// LS Electric XG5000 project: xg
// PLC NewPLC
// module base 0 slot 0: 입출력 모듈:XBC-DR32H (DC 24V 입력, 릴레이 출력 32점)
// module base 0 slot 1: 위치결정 모듈:XBF-PD02A (위치결정 펄스(LD)출력형, 2축)
// module base 0 slot 2: 출력 모듈:XBE-TN/TP16A (트랜지스터 출력, 16점 (싱크출력/소스출력))

PROGRAM NewProgram (task: 스캔 프로그램)

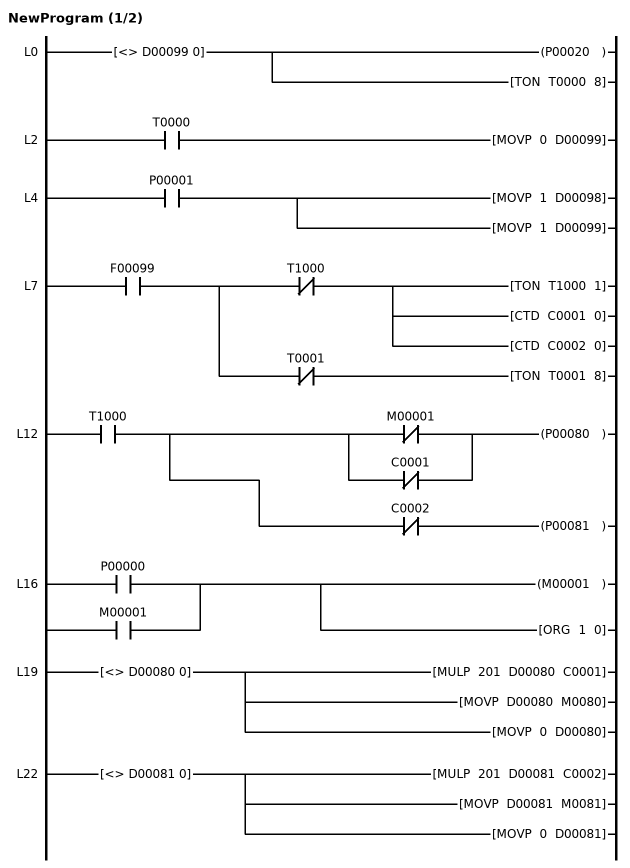
; L0
LOAD<>    D00099 0
OUT       P00020
TON       T0000 8
; L2
LOAD      T0000
MOVP      0 D00099
; L4
LOAD      P00001
MOVP      1 D00098
MOVP      1 D00099
; L7
LOAD      F00099
MPUSH
AND NOT   T1000
TON       T1000 1
CTD       C0001 0
CTD       C0002 0
MPOP
AND NOT   T0001
TON       T0001 8
; L12
LOAD      T1000
MPUSH
LOAD NOT  M00001
OR NOT    C0001
AND LOAD
OUT       P00080
MPOP
AND NOT   C0002
OUT       P00081
; L16
LOAD      P00000
OR        M00001
OUT       M00001
ORG       1 0
; L19
LOAD<>    D00080 0
MULP      201 D00080 C0001
MOVP      D00080 M0080
MOVP      0 D00080
; L22
LOAD<>    D00081 0
MULP      201 D00081 C0002
MOVP      D00081 M0081
MOVP      0 D00081

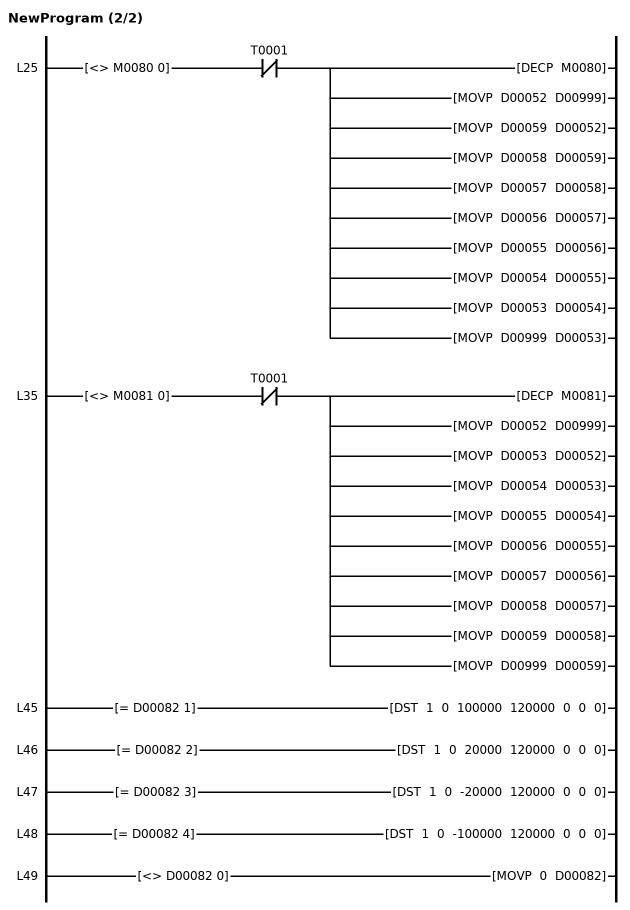
; L25
LOAD<>    M0080 0
AND NOT   T0001
DECP      M0080
MOVP      D00052 D00999
MOVP      D00059 D00052
MOVP      D00058 D00059
MOVP      D00057 D00058
MOVP      D00056 D00057
MOVP      D00055 D00056
MOVP      D00054 D00055
MOVP      D00053 D00054
MOVP      D00999 D00053
; L35
LOAD<>    M0081 0
AND NOT   T0001
DECP      M0081
MOVP      D00052 D00999
MOVP      D00053 D00052
MOVP      D00054 D00053
MOVP      D00055 D00054
MOVP      D00056 D00055
MOVP      D00057 D00056
MOVP      D00058 D00057
MOVP      D00059 D00058
MOVP      D00999 D00059
; L45
LOAD=     D00082 1
DST       1 0 100000 120000 0 0 0
; L46
LOAD=     D00082 2
DST       1 0 20000 120000 0 0 0
; L47
LOAD=     D00082 3
DST       1 0 -20000 120000 0 0 0
; L48
LOAD=     D00082 4
DST       1 0 -100000 120000 0 0 0
; L49
LOAD<>    D00082 0
MOVP      0 D00082